TYPE ST_Motor :
STRUCT
	Axis        : AXIS_REF;   // Axis reference (default to all motors)
    bEnable     : BOOL;       // Enable command
    bReset      : BOOL;       // Reset command
    bError      : BOOL;       // Error flag
    nErrorID    : UDINT;      // Error ID
    bBusy       : BOOL;       // In moviment state
    bInPosition : BOOL;       // Indicates when the position was reached
	rActualPosition : LREAL;  // Show de actual motor position
	
	// Additional variables to direct link (%I e %Q):
    nState        	AT %I*	: UINT;	 //Actual State (Axis StatusWord)
    nControlWord  	AT %Q*	: UINT;	 //Control Word (ControlWord send to axis)
    rActualPos 		AT %I*	: LREAL; //Real Actual Axis Position (Position Actual Value)
	rActualTorque	AT %I*	: LREAL; //Real Actual Axis Torque (Torque Actual Value)
    rActualVel 		AT %I*	: LREAL; //Real Actual Axis Velocity (Velocity Actual Value)
	iOperational	AT %I*	: BOOL;
	iHomed			AT %I*	: BOOL;
	iNotMoving		AT %I*	: BOOL;
	iError			AT %I*	: BOOL;
	nErrorCode		AT %I*	: UDINT;
	bMotionCommandsLocked	AT %I*	: BOOL;
	
END_STRUCT
END_TYPE

(* stored: Version 1.1.0.1, ProductVersion 3.1.4024.15
   DUT ST_Motor: Id {2c3c1834-2f58-41c6-810f-8bd283ecb8c2} *)
